TYPE ST_MovisafeCSSx1a_Config :
STRUCT	
	bSwapProcessData		: BOOL; //SWAP Process Data from/to FIELDBUS
END_STRUCT
END_TYPE

(* stored: Version 1.1.0.1, ProductVersion 3.1.4024.12
   DUT ST_MovisafeCSSx1a_Config: Id {8511d0ac-9b64-0794-3fcf-731ce4a07f75} *)
